// Contains CoE indexes and sub indexes for Bronkhorst EtherCAT mass flow controller
TYPE ST_ControllerCoeList :
STRUCT
	FluidName		: ZigaLibs_Core.ST_CoeEntry_String30 	:= (Index := 16#2001, SubIndex := 16#12);
	Capacity 		: ZigaLibs_Core.ST_CoeEntry_REAL 		:= (Index := 16#2001, SubIndex := 16#0E);
	CapacityUnit 	: ZigaLibs_Core.ST_CoeEntry_String30 	:= (Index := 16#2001, SubIndex := 16#20);
	DecimalDigits 	: ZigaLibs_Core.ST_CoeEntry_INT 		:= (Index := 16#6407, SubIndex := 16#01);
	ControlMode 	: ZigaLibs_Core.ST_CoeEntry_USINT 		:= (Index := 16#6423, SubIndex := 16#01);
	ControllerSpeed	: ZigaLibs_Core.ST_CoeEntry_USINT		:= (Index := 16#2072, Subindex := 16#1F);
END_STRUCT
END_TYPE

(* stored: Version 1.1.0.1, ProductVersion 3.1.4024.16
   DUT ST_ControllerCoeList: Id {07592a42-9fc5-0eb9-1f52-2c09efd9255d} *)
